// TIA Portal V19 export
FUNCTION "mfg filtration LOGIC" : Void   // FC8, LAD
{ S7_Optimized_Access := 'TRUE' }
// stored: SetENOAutomatically false
   VAR_TEMP   // added for the SCL form of the ladder/FBD networks
      _w1 : Bool;
   END_VAR
BEGIN

REGION Network 1: MFG PROCESS START
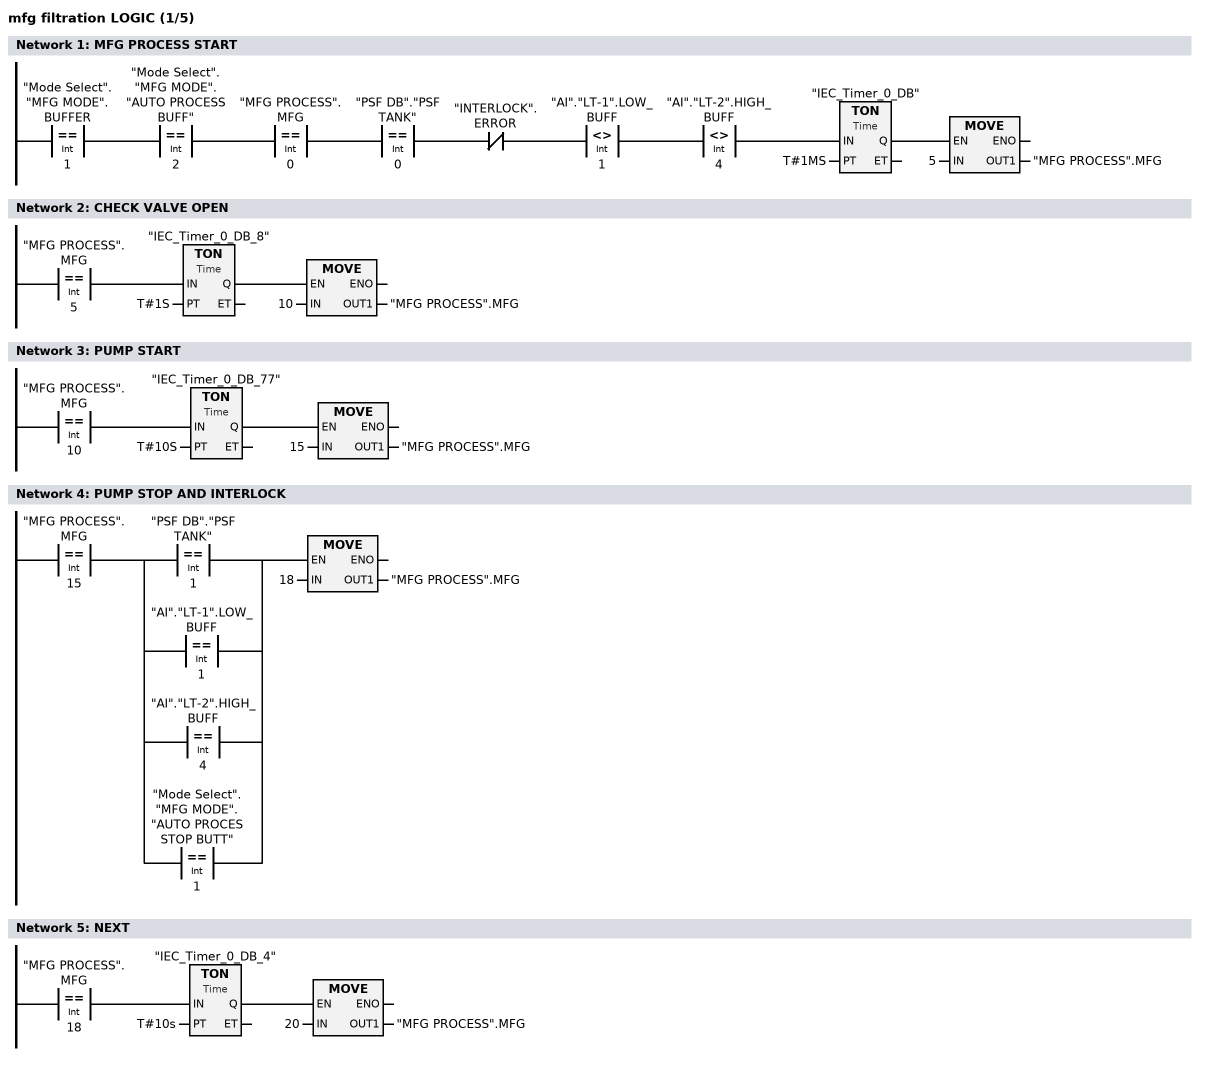
   RUNG wire#powerrail
      { S7_Templates := "SrcType := Int" } EQ_Contact(in1 := "Mode Select"."MFG MODE".BUFFER, in2 := 1)
      { S7_Templates := "SrcType := Int" } EQ_Contact(in1 := "Mode Select"."MFG MODE"."AUTO PROCESS BUFF", in2 := 2)
      { S7_Templates := "SrcType := Int" } EQ_Contact(in1 := "MFG PROCESS".MFG, in2 := 0)
      { S7_Templates := "SrcType := Int" } EQ_Contact(in1 := "PSF DB"."PSF TANK", in2 := 0)
      I_Contact( "INTERLOCK".ERROR )
      { S7_Templates := "SrcType := Int" } NE_Contact(in1 := "AI"."LT-1".LOW_BUFF, in2 := 1)
      { S7_Templates := "SrcType := Int" } NE_Contact(in1 := "AI"."LT-2".HIGH_BUFF, in2 := 4)
      { S7_Templates := "time_type := Time" } "IEC_Timer_0_DB".TON(pt := T#1MS, et =>)
      Move(in := 5, out1 => "MFG PROCESS".MFG)
   END_RUNG
   // the same network as SCL:
   "IEC_Timer_0_DB".TON(IN := ("Mode Select"."MFG MODE".BUFFER = 1) AND ("Mode Select"."MFG MODE"."AUTO PROCESS BUFF" = 2) AND ("MFG PROCESS".MFG = 0) AND ("PSF DB"."PSF TANK" = 0) AND NOT "INTERLOCK".ERROR AND ("AI"."LT-1".LOW_BUFF <> 1) AND ("AI"."LT-2".HIGH_BUFF <> 4),
                        PT := T#1MS);
   IF "IEC_Timer_0_DB".Q THEN "MFG PROCESS".MFG := 5; END_IF;
END_REGION

REGION Network 2: CHECK VALVE OPEN
   RUNG wire#powerrail
      { S7_Templates := "SrcType := Int" } EQ_Contact(in1 := "MFG PROCESS".MFG, in2 := 5)
      { S7_Templates := "time_type := Time" } "IEC_Timer_0_DB_8".TON(pt := T#1S, et =>)
      Move(in := 10, out1 => "MFG PROCESS".MFG)
   END_RUNG
   // the same network as SCL:
   "IEC_Timer_0_DB_8".TON(IN := "MFG PROCESS".MFG = 5, PT := T#1S);
   IF "IEC_Timer_0_DB_8".Q THEN "MFG PROCESS".MFG := 10; END_IF;
END_REGION

REGION Network 3: PUMP START
   RUNG wire#powerrail
      { S7_Templates := "SrcType := Int" } EQ_Contact(in1 := "MFG PROCESS".MFG, in2 := 10)
      { S7_Templates := "time_type := Time" } "IEC_Timer_0_DB_77".TON(pt := T#10S, et =>)
      Move(in := 15, out1 => "MFG PROCESS".MFG)
   END_RUNG
   // the same network as SCL:
   "IEC_Timer_0_DB_77".TON(IN := "MFG PROCESS".MFG = 10, PT := T#10S);
   IF "IEC_Timer_0_DB_77".Q THEN "MFG PROCESS".MFG := 15; END_IF;
END_REGION

REGION Network 4: PUMP STOP AND INTERLOCK
   RUNG wire#powerrail
      { S7_Templates := "SrcType := Int" } EQ_Contact(in1 := "MFG PROCESS".MFG, in2 := 15)
      wire#w1
      { S7_Templates := "SrcType := Int" } EQ_Contact(in1 := "PSF DB"."PSF TANK", in2 := 1)
      wire#w2
      Move(in := 18, out1 => "MFG PROCESS".MFG)
   END_RUNG
   RUNG wire#w1
      { S7_Templates := "SrcType := Int" } EQ_Contact(in1 := "AI"."LT-1".LOW_BUFF, in2 := 1)
   END_RUNG wire#w2
   RUNG wire#w1
      { S7_Templates := "SrcType := Int" } EQ_Contact(in1 := "AI"."LT-2".HIGH_BUFF, in2 := 4)
   END_RUNG wire#w2
   RUNG wire#w1
      { S7_Templates := "SrcType := Int" } EQ_Contact(in1 := "Mode Select"."MFG MODE"."AUTO PROCES STOP BUTT", in2 := 1)
   END_RUNG wire#w2
   // the same network as SCL:
   IF ("MFG PROCESS".MFG = 15) AND (("PSF DB"."PSF TANK" = 1) OR ("AI"."LT-1".LOW_BUFF = 1) OR ("AI"."LT-2".HIGH_BUFF = 4) OR ("Mode Select"."MFG MODE"."AUTO PROCES STOP BUTT" = 1)) THEN
       "MFG PROCESS".MFG := 18;
   END_IF;
END_REGION

REGION Network 5: NEXT
   RUNG wire#powerrail
      { S7_Templates := "SrcType := Int" } EQ_Contact(in1 := "MFG PROCESS".MFG, in2 := 18)
      { S7_Templates := "time_type := Time" } "IEC_Timer_0_DB_4".TON(pt := T#10s, et =>)
      Move(in := 20, out1 => "MFG PROCESS".MFG)
   END_RUNG
   // the same network as SCL:
   "IEC_Timer_0_DB_4".TON(IN := "MFG PROCESS".MFG = 18, PT := T#10s);
   IF "IEC_Timer_0_DB_4".Q THEN "MFG PROCESS".MFG := 20; END_IF;
END_REGION

REGION Network 6: MFG PROCESS OVER
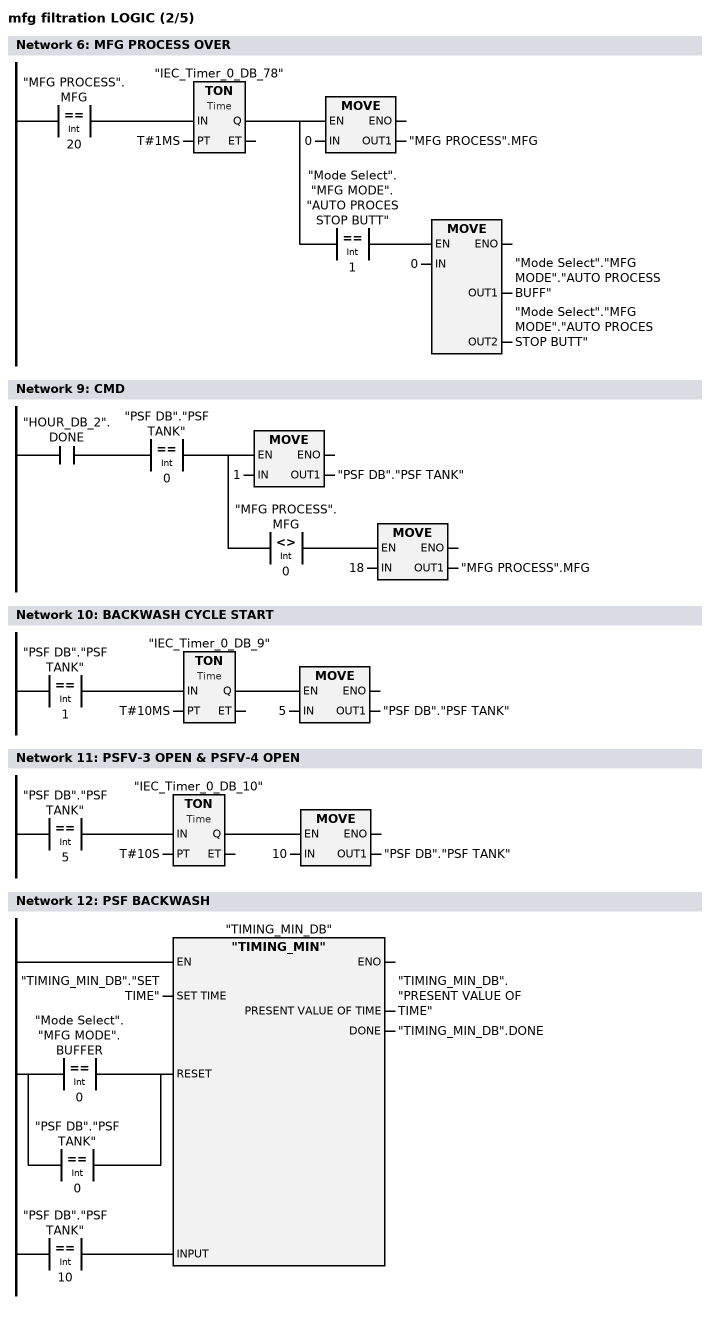
   RUNG wire#powerrail
      { S7_Templates := "SrcType := Int" } EQ_Contact(in1 := "MFG PROCESS".MFG, in2 := 20)
      { S7_Templates := "time_type := Time" } "IEC_Timer_0_DB_78".TON(pt := T#1MS, et =>)
      wire#w1
      Move(in := 0, out1 => "MFG PROCESS".MFG)
   END_RUNG
   RUNG wire#w1
      { S7_Templates := "SrcType := Int" } EQ_Contact(in1 := "Mode Select"."MFG MODE"."AUTO PROCES STOP BUTT", in2 := 1)
      Move(in := 0, out1 => "Mode Select"."MFG MODE"."AUTO PROCESS BUFF", out2 => "Mode Select"."MFG MODE"."AUTO PROCES STOP BUTT")
   END_RUNG
   // the same network as SCL:
   "IEC_Timer_0_DB_78".TON(IN := "MFG PROCESS".MFG = 20, PT := T#1MS);
   IF "IEC_Timer_0_DB_78".Q THEN "MFG PROCESS".MFG := 0; END_IF;
   IF "IEC_Timer_0_DB_78".Q AND ("Mode Select"."MFG MODE"."AUTO PROCES STOP BUTT" = 1) THEN
       "Mode Select"."MFG MODE"."AUTO PROCESS BUFF" := 0;
       "Mode Select"."MFG MODE"."AUTO PROCES STOP BUTT" := 0;
   END_IF;
END_REGION

REGION Network 9: CMD
   RUNG wire#powerrail
      Contact( "HOUR_DB_2".DONE )
      { S7_Templates := "SrcType := Int" } EQ_Contact(in1 := "PSF DB"."PSF TANK", in2 := 0)
      wire#w1
      Move(in := 1, out1 => "PSF DB"."PSF TANK")
   END_RUNG
   RUNG wire#w1
      { S7_Templates := "SrcType := Int" } NE_Contact(in1 := "MFG PROCESS".MFG, in2 := 0)
      Move(in := 18, out1 => "MFG PROCESS".MFG)
   END_RUNG
   // the same network as SCL:
   #_w1 := "HOUR_DB_2".DONE AND ("PSF DB"."PSF TANK" = 0);
   IF #_w1 THEN "PSF DB"."PSF TANK" := 1; END_IF;
   IF #_w1 AND ("MFG PROCESS".MFG <> 0) THEN "MFG PROCESS".MFG := 18; END_IF;
END_REGION

REGION Network 10: BACKWASH CYCLE START
   RUNG wire#powerrail
      { S7_Templates := "SrcType := Int" } EQ_Contact(in1 := "PSF DB"."PSF TANK", in2 := 1)
      { S7_Templates := "time_type := Time" } "IEC_Timer_0_DB_9".TON(pt := T#10MS, et =>)
      Move(in := 5, out1 => "PSF DB"."PSF TANK")
   END_RUNG
   // the same network as SCL:
   "IEC_Timer_0_DB_9".TON(IN := "PSF DB"."PSF TANK" = 1, PT := T#10MS);
   IF "IEC_Timer_0_DB_9".Q THEN "PSF DB"."PSF TANK" := 5; END_IF;
END_REGION

REGION Network 11: PSFV-3 OPEN & PSFV-4 OPEN
   RUNG wire#powerrail
      { S7_Templates := "SrcType := Int" } EQ_Contact(in1 := "PSF DB"."PSF TANK", in2 := 5)
      { S7_Templates := "time_type := Time" } "IEC_Timer_0_DB_10".TON(pt := T#10S, et =>)
      Move(in := 10, out1 => "PSF DB"."PSF TANK")
   END_RUNG
   // the same network as SCL:
   "IEC_Timer_0_DB_10".TON(IN := "PSF DB"."PSF TANK" = 5, PT := T#10S);
   IF "IEC_Timer_0_DB_10".Q THEN "PSF DB"."PSF TANK" := 10; END_IF;
END_REGION

REGION Network 12: PSF BACKWASH
   RUNG wire#powerrail
      "TIMING_MIN_DB"(RESET := wire#w1, INPUT := wire#w2, "SET TIME" := "TIMING_MIN_DB"."SET TIME", "PRESENT VALUE OF TIME" => "TIMING_MIN_DB"."PRESENT VALUE OF TIME", DONE => "TIMING_MIN_DB".DONE)
   END_RUNG
   RUNG wire#powerrail
      { S7_Templates := "SrcType := Int" } EQ_Contact(in1 := "Mode Select"."MFG MODE".BUFFER, in2 := 0)
   END_RUNG wire#w1
   RUNG wire#powerrail
      { S7_Templates := "SrcType := Int" } EQ_Contact(in1 := "PSF DB"."PSF TANK", in2 := 0)
   END_RUNG wire#w1
   RUNG wire#powerrail
      { S7_Templates := "SrcType := Int" } EQ_Contact(in1 := "PSF DB"."PSF TANK", in2 := 10)
   END_RUNG wire#w2
   // the same network as SCL:
   "TIMING_MIN_DB"("SET TIME" := "TIMING_MIN_DB"."SET TIME",   // "TIMING_MIN"
                   RESET := ("Mode Select"."MFG MODE".BUFFER = 0) OR ("PSF DB"."PSF TANK" = 0),
                   INPUT := "PSF DB"."PSF TANK" = 10,
                   "PRESENT VALUE OF TIME" => "TIMING_MIN_DB"."PRESENT VALUE OF TIME",
                   DONE => "TIMING_MIN_DB".DONE);
END_REGION

REGION Network 13: TIMER DONE
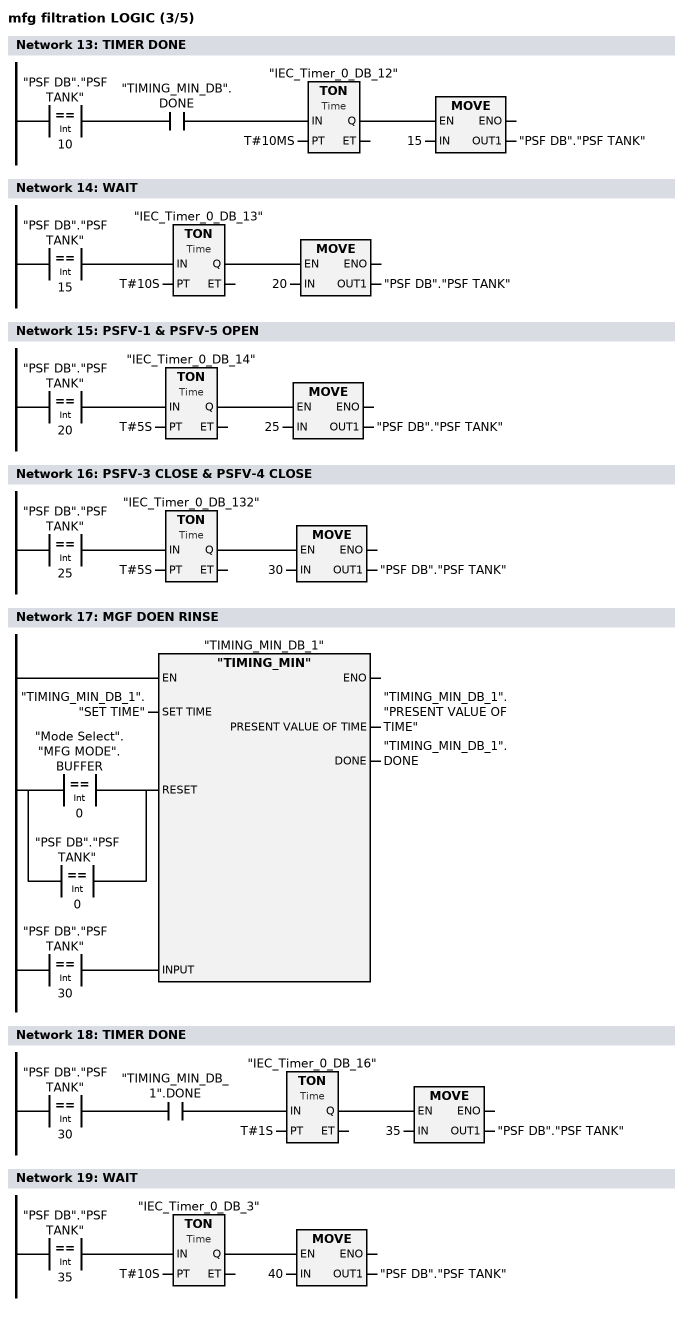
   RUNG wire#powerrail
      { S7_Templates := "SrcType := Int" } EQ_Contact(in1 := "PSF DB"."PSF TANK", in2 := 10)
      Contact( "TIMING_MIN_DB".DONE )
      { S7_Templates := "time_type := Time" } "IEC_Timer_0_DB_12".TON(pt := T#10MS, et =>)
      Move(in := 15, out1 => "PSF DB"."PSF TANK")
   END_RUNG
   // the same network as SCL:
   "IEC_Timer_0_DB_12".TON(IN := ("PSF DB"."PSF TANK" = 10) AND "TIMING_MIN_DB".DONE, PT := T#10MS);
   IF "IEC_Timer_0_DB_12".Q THEN "PSF DB"."PSF TANK" := 15; END_IF;
END_REGION

REGION Network 14: WAIT
   RUNG wire#powerrail
      { S7_Templates := "SrcType := Int" } EQ_Contact(in1 := "PSF DB"."PSF TANK", in2 := 15)
      { S7_Templates := "time_type := Time" } "IEC_Timer_0_DB_13".TON(pt := T#10S, et =>)
      Move(in := 20, out1 => "PSF DB"."PSF TANK")
   END_RUNG
   // the same network as SCL:
   "IEC_Timer_0_DB_13".TON(IN := "PSF DB"."PSF TANK" = 15, PT := T#10S);
   IF "IEC_Timer_0_DB_13".Q THEN "PSF DB"."PSF TANK" := 20; END_IF;
END_REGION

REGION Network 15: PSFV-1 & PSFV-5 OPEN
   RUNG wire#powerrail
      { S7_Templates := "SrcType := Int" } EQ_Contact(in1 := "PSF DB"."PSF TANK", in2 := 20)
      { S7_Templates := "time_type := Time" } "IEC_Timer_0_DB_14".TON(pt := T#5S, et =>)
      Move(in := 25, out1 => "PSF DB"."PSF TANK")
   END_RUNG
   // the same network as SCL:
   "IEC_Timer_0_DB_14".TON(IN := "PSF DB"."PSF TANK" = 20, PT := T#5S);
   IF "IEC_Timer_0_DB_14".Q THEN "PSF DB"."PSF TANK" := 25; END_IF;
END_REGION

REGION Network 16: PSFV-3 CLOSE & PSFV-4 CLOSE
   RUNG wire#powerrail
      { S7_Templates := "SrcType := Int" } EQ_Contact(in1 := "PSF DB"."PSF TANK", in2 := 25)
      { S7_Templates := "time_type := Time" } "IEC_Timer_0_DB_132".TON(pt := T#5S, et =>)
      Move(in := 30, out1 => "PSF DB"."PSF TANK")
   END_RUNG
   // the same network as SCL:
   "IEC_Timer_0_DB_132".TON(IN := "PSF DB"."PSF TANK" = 25, PT := T#5S);
   IF "IEC_Timer_0_DB_132".Q THEN "PSF DB"."PSF TANK" := 30; END_IF;
END_REGION

REGION Network 17: MGF DOEN RINSE
   RUNG wire#powerrail
      "TIMING_MIN_DB_1"(RESET := wire#w1, INPUT := wire#w2, "SET TIME" := "TIMING_MIN_DB_1"."SET TIME", "PRESENT VALUE OF TIME" => "TIMING_MIN_DB_1"."PRESENT VALUE OF TIME", DONE => "TIMING_MIN_DB_1".DONE)
   END_RUNG
   RUNG wire#powerrail
      { S7_Templates := "SrcType := Int" } EQ_Contact(in1 := "Mode Select"."MFG MODE".BUFFER, in2 := 0)
   END_RUNG wire#w1
   RUNG wire#powerrail
      { S7_Templates := "SrcType := Int" } EQ_Contact(in1 := "PSF DB"."PSF TANK", in2 := 0)
   END_RUNG wire#w1
   RUNG wire#powerrail
      { S7_Templates := "SrcType := Int" } EQ_Contact(in1 := "PSF DB"."PSF TANK", in2 := 30)
   END_RUNG wire#w2
   // the same network as SCL:
   "TIMING_MIN_DB_1"("SET TIME" := "TIMING_MIN_DB_1"."SET TIME",   // "TIMING_MIN"
                     RESET := ("Mode Select"."MFG MODE".BUFFER = 0) OR ("PSF DB"."PSF TANK" = 0),
                     INPUT := "PSF DB"."PSF TANK" = 30,
                     "PRESENT VALUE OF TIME" => "TIMING_MIN_DB_1"."PRESENT VALUE OF TIME",
                     DONE => "TIMING_MIN_DB_1".DONE);
END_REGION

REGION Network 18: TIMER DONE
   RUNG wire#powerrail
      { S7_Templates := "SrcType := Int" } EQ_Contact(in1 := "PSF DB"."PSF TANK", in2 := 30)
      Contact( "TIMING_MIN_DB_1".DONE )
      { S7_Templates := "time_type := Time" } "IEC_Timer_0_DB_16".TON(pt := T#1S, et =>)
      Move(in := 35, out1 => "PSF DB"."PSF TANK")
   END_RUNG
   // the same network as SCL:
   "IEC_Timer_0_DB_16".TON(IN := ("PSF DB"."PSF TANK" = 30) AND "TIMING_MIN_DB_1".DONE, PT := T#1S);
   IF "IEC_Timer_0_DB_16".Q THEN "PSF DB"."PSF TANK" := 35; END_IF;
END_REGION

REGION Network 19: WAIT
   RUNG wire#powerrail
      { S7_Templates := "SrcType := Int" } EQ_Contact(in1 := "PSF DB"."PSF TANK", in2 := 35)
      { S7_Templates := "time_type := Time" } "IEC_Timer_0_DB_3".TON(pt := T#10S, et =>)
      Move(in := 40, out1 => "PSF DB"."PSF TANK")
   END_RUNG
   // the same network as SCL:
   "IEC_Timer_0_DB_3".TON(IN := "PSF DB"."PSF TANK" = 35, PT := T#10S);
   IF "IEC_Timer_0_DB_3".Q THEN "PSF DB"."PSF TANK" := 40; END_IF;
END_REGION

REGION Network 20: PSFV1 & PSFV2 & ACFV3 & ACFV4 OPEN
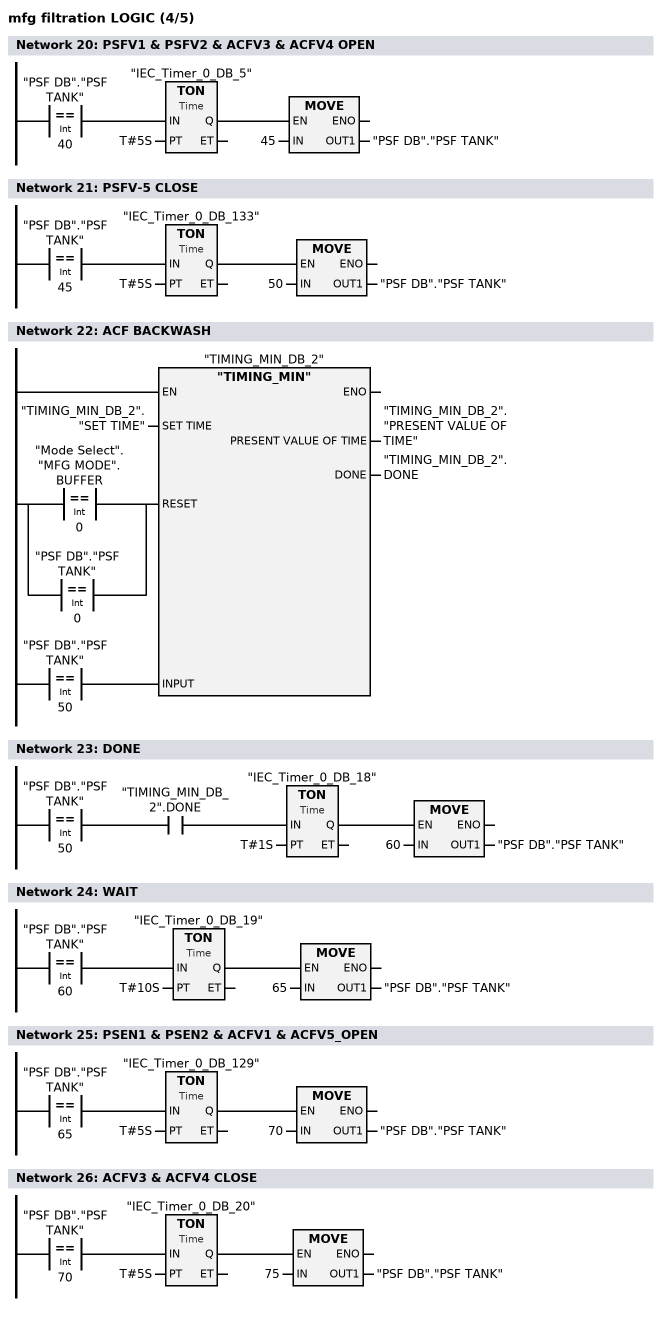
   RUNG wire#powerrail
      { S7_Templates := "SrcType := Int" } EQ_Contact(in1 := "PSF DB"."PSF TANK", in2 := 40)
      { S7_Templates := "time_type := Time" } "IEC_Timer_0_DB_5".TON(pt := T#5S, et =>)
      Move(in := 45, out1 => "PSF DB"."PSF TANK")
   END_RUNG
   // the same network as SCL:
   "IEC_Timer_0_DB_5".TON(IN := "PSF DB"."PSF TANK" = 40, PT := T#5S);
   IF "IEC_Timer_0_DB_5".Q THEN "PSF DB"."PSF TANK" := 45; END_IF;
END_REGION

REGION Network 21: PSFV-5 CLOSE
   RUNG wire#powerrail
      { S7_Templates := "SrcType := Int" } EQ_Contact(in1 := "PSF DB"."PSF TANK", in2 := 45)
      { S7_Templates := "time_type := Time" } "IEC_Timer_0_DB_133".TON(pt := T#5S, et =>)
      Move(in := 50, out1 => "PSF DB"."PSF TANK")
   END_RUNG
   // the same network as SCL:
   "IEC_Timer_0_DB_133".TON(IN := "PSF DB"."PSF TANK" = 45, PT := T#5S);
   IF "IEC_Timer_0_DB_133".Q THEN "PSF DB"."PSF TANK" := 50; END_IF;
END_REGION

REGION Network 22: ACF BACKWASH
   RUNG wire#powerrail
      "TIMING_MIN_DB_2"(RESET := wire#w1, INPUT := wire#w2, "SET TIME" := "TIMING_MIN_DB_2"."SET TIME", "PRESENT VALUE OF TIME" => "TIMING_MIN_DB_2"."PRESENT VALUE OF TIME", DONE => "TIMING_MIN_DB_2".DONE)
   END_RUNG
   RUNG wire#powerrail
      { S7_Templates := "SrcType := Int" } EQ_Contact(in1 := "Mode Select"."MFG MODE".BUFFER, in2 := 0)
   END_RUNG wire#w1
   RUNG wire#powerrail
      { S7_Templates := "SrcType := Int" } EQ_Contact(in1 := "PSF DB"."PSF TANK", in2 := 0)
   END_RUNG wire#w1
   RUNG wire#powerrail
      { S7_Templates := "SrcType := Int" } EQ_Contact(in1 := "PSF DB"."PSF TANK", in2 := 50)
   END_RUNG wire#w2
   // the same network as SCL:
   "TIMING_MIN_DB_2"("SET TIME" := "TIMING_MIN_DB_2"."SET TIME",   // "TIMING_MIN"
                     RESET := ("Mode Select"."MFG MODE".BUFFER = 0) OR ("PSF DB"."PSF TANK" = 0),
                     INPUT := "PSF DB"."PSF TANK" = 50,
                     "PRESENT VALUE OF TIME" => "TIMING_MIN_DB_2"."PRESENT VALUE OF TIME",
                     DONE => "TIMING_MIN_DB_2".DONE);
END_REGION

REGION Network 23: DONE
   RUNG wire#powerrail
      { S7_Templates := "SrcType := Int" } EQ_Contact(in1 := "PSF DB"."PSF TANK", in2 := 50)
      Contact( "TIMING_MIN_DB_2".DONE )
      { S7_Templates := "time_type := Time" } "IEC_Timer_0_DB_18".TON(pt := T#1S, et =>)
      Move(in := 60, out1 => "PSF DB"."PSF TANK")
   END_RUNG
   // the same network as SCL:
   "IEC_Timer_0_DB_18".TON(IN := ("PSF DB"."PSF TANK" = 50) AND "TIMING_MIN_DB_2".DONE, PT := T#1S);
   IF "IEC_Timer_0_DB_18".Q THEN "PSF DB"."PSF TANK" := 60; END_IF;
END_REGION

REGION Network 24: WAIT
   RUNG wire#powerrail
      { S7_Templates := "SrcType := Int" } EQ_Contact(in1 := "PSF DB"."PSF TANK", in2 := 60)
      { S7_Templates := "time_type := Time" } "IEC_Timer_0_DB_19".TON(pt := T#10S, et =>)
      Move(in := 65, out1 => "PSF DB"."PSF TANK")
   END_RUNG
   // the same network as SCL:
   "IEC_Timer_0_DB_19".TON(IN := "PSF DB"."PSF TANK" = 60, PT := T#10S);
   IF "IEC_Timer_0_DB_19".Q THEN "PSF DB"."PSF TANK" := 65; END_IF;
END_REGION

REGION Network 25: PSEN1 & PSEN2 & ACFV1 & ACFV5_OPEN
   RUNG wire#powerrail
      { S7_Templates := "SrcType := Int" } EQ_Contact(in1 := "PSF DB"."PSF TANK", in2 := 65)
      { S7_Templates := "time_type := Time" } "IEC_Timer_0_DB_129".TON(pt := T#5S, et =>)
      Move(in := 70, out1 => "PSF DB"."PSF TANK")
   END_RUNG
   // the same network as SCL:
   "IEC_Timer_0_DB_129".TON(IN := "PSF DB"."PSF TANK" = 65, PT := T#5S);
   IF "IEC_Timer_0_DB_129".Q THEN "PSF DB"."PSF TANK" := 70; END_IF;
END_REGION

REGION Network 26: ACFV3 & ACFV4 CLOSE
   RUNG wire#powerrail
      { S7_Templates := "SrcType := Int" } EQ_Contact(in1 := "PSF DB"."PSF TANK", in2 := 70)
      { S7_Templates := "time_type := Time" } "IEC_Timer_0_DB_20".TON(pt := T#5S, et =>)
      Move(in := 75, out1 => "PSF DB"."PSF TANK")
   END_RUNG
   // the same network as SCL:
   "IEC_Timer_0_DB_20".TON(IN := "PSF DB"."PSF TANK" = 70, PT := T#5S);
   IF "IEC_Timer_0_DB_20".Q THEN "PSF DB"."PSF TANK" := 75; END_IF;
END_REGION

REGION Network 27: ACF DOWN RINSE
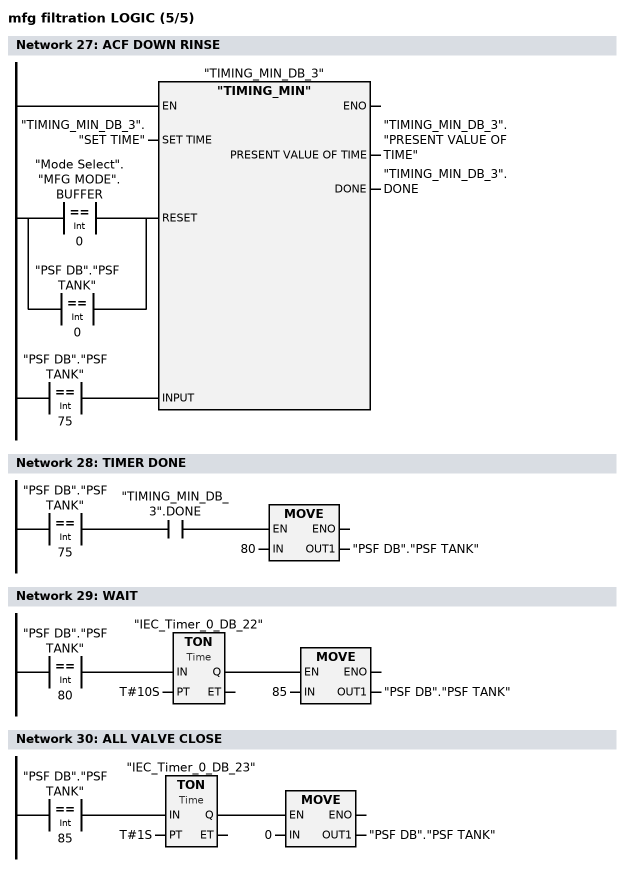
   RUNG wire#powerrail
      "TIMING_MIN_DB_3"(RESET := wire#w1, INPUT := wire#w2, "SET TIME" := "TIMING_MIN_DB_3"."SET TIME", "PRESENT VALUE OF TIME" => "TIMING_MIN_DB_3"."PRESENT VALUE OF TIME", DONE => "TIMING_MIN_DB_3".DONE)
   END_RUNG
   RUNG wire#powerrail
      { S7_Templates := "SrcType := Int" } EQ_Contact(in1 := "Mode Select"."MFG MODE".BUFFER, in2 := 0)
   END_RUNG wire#w1
   RUNG wire#powerrail
      { S7_Templates := "SrcType := Int" } EQ_Contact(in1 := "PSF DB"."PSF TANK", in2 := 0)
   END_RUNG wire#w1
   RUNG wire#powerrail
      { S7_Templates := "SrcType := Int" } EQ_Contact(in1 := "PSF DB"."PSF TANK", in2 := 75)
   END_RUNG wire#w2
   // the same network as SCL:
   "TIMING_MIN_DB_3"("SET TIME" := "TIMING_MIN_DB_3"."SET TIME",   // "TIMING_MIN"
                     RESET := ("Mode Select"."MFG MODE".BUFFER = 0) OR ("PSF DB"."PSF TANK" = 0),
                     INPUT := "PSF DB"."PSF TANK" = 75,
                     "PRESENT VALUE OF TIME" => "TIMING_MIN_DB_3"."PRESENT VALUE OF TIME",
                     DONE => "TIMING_MIN_DB_3".DONE);
END_REGION

REGION Network 28: TIMER DONE
   RUNG wire#powerrail
      { S7_Templates := "SrcType := Int" } EQ_Contact(in1 := "PSF DB"."PSF TANK", in2 := 75)
      Contact( "TIMING_MIN_DB_3".DONE )
      Move(in := 80, out1 => "PSF DB"."PSF TANK")
   END_RUNG
   // the same network as SCL:
   IF ("PSF DB"."PSF TANK" = 75) AND "TIMING_MIN_DB_3".DONE THEN "PSF DB"."PSF TANK" := 80; END_IF;
END_REGION

REGION Network 29: WAIT
   RUNG wire#powerrail
      { S7_Templates := "SrcType := Int" } EQ_Contact(in1 := "PSF DB"."PSF TANK", in2 := 80)
      { S7_Templates := "time_type := Time" } "IEC_Timer_0_DB_22".TON(pt := T#10S, et =>)
      Move(in := 85, out1 => "PSF DB"."PSF TANK")
   END_RUNG
   // the same network as SCL:
   "IEC_Timer_0_DB_22".TON(IN := "PSF DB"."PSF TANK" = 80, PT := T#10S);
   IF "IEC_Timer_0_DB_22".Q THEN "PSF DB"."PSF TANK" := 85; END_IF;
END_REGION

REGION Network 30: ALL VALVE CLOSE
   RUNG wire#powerrail
      { S7_Templates := "SrcType := Int" } EQ_Contact(in1 := "PSF DB"."PSF TANK", in2 := 85)
      { S7_Templates := "time_type := Time" } "IEC_Timer_0_DB_23".TON(pt := T#1S, et =>)
      Move(in := 0, out1 => "PSF DB"."PSF TANK")
   END_RUNG
   // the same network as SCL:
   "IEC_Timer_0_DB_23".TON(IN := "PSF DB"."PSF TANK" = 85, PT := T#1S);
   IF "IEC_Timer_0_DB_23".Q THEN "PSF DB"."PSF TANK" := 0; END_IF;
END_REGION
END_FUNCTION
